FUNCTION_BLOCK FB_DIVIDE
VAR_INPUT
	inValue01:REAL;
	inValue02:REAL;
END_VAR
VAR_OUTPUT
	outSum:REAL;
END_VAR
VAR
	Val01_Local:REAL;
	Val02_Local:REAL;
	Sum_Local:REAL;
END_VAR

Val01_Local:=inValue01;
Val02_Local:=inValue02;

IF inValue02=0 THEN ;
	ELSE Sum_Local:=Val01_Local/Val02_Local;
END_IF

outSum:=Sum_Local;

END_FUNCTION_BLOCK

(* stored: Version 1.1.0.1, ProductVersion 3.1.4024.4
   POU FB_DIVIDE: Id {b520a7dc-505f-44df-ad4c-429d6c9dfa61}, SpecialFunc None *)
